{attribute 'GeneratedUsingTerminal: EK1100-0000-0018'}
{attribute addProperty BoxType "EK1100-0000-0018"}
{attribute addProperty Id "Beckhoff_EL73xxEK1122Beckhoff_EL73xxEK1122_D359B3E92A_0001_EL7332_0000_0016EL7332_B885ACFD38A_0002_EL7332_0000_0017EL7332_B885ACFD38A_0003_EL7332_0000_0018EL7332_B885ACFD38A_0004_EL7332_0000_0019EL7332_B885ACFD38A_0005_EL7332_0000_0020EL7332_B885ACFD38A_0006_EL7332_0000_0021EL7332_B885ACFD38A_0007_EL7332_0000_0022EL7332_B885ACFD38A_0008_EL7332_0000_0023EL7332_B885ACFD38A_0009_EL7332_0000_0024EL7332_B885ACFD38A_0010_EL7342_0000_0016EL7342_A970B60778A_0011_EL7342_0000_0017EL7342_A970B60778A_0012_EL7342_0000_0018EL7342_A970B60778A_0013_EL7342_0000_0019EL7342_A970B60778A_0014_EL7342_0000_0020EL7342_A970B60778A_0015_EL7342_0000_0021EL7342_A970B60778A_0016_EL7342_0000_0022EL7342_A970B60778A_0017_EL7342_0000_0023EL7342_C56E195380A_0018_EL7342_0035_0019EL7342_A970B60778A_0019_EL7342_0035_0020EL7342_A970B60778"}
{attribute addProperty CRC "3215524844"}
{attribute addProperty Size "1126"}
TYPE Beckhoff_EL73xx_BFA903EC EXTENDS EK1100_1FC0878B :
STRUCT
	{attribute addProperty Name "Beckhoff_EL73xxEK1122"}
	{attribute addProperty PreviousPort "Beckhoff EL73xx : B"}
	Beckhoff_EL73xxEK1122 : Beckhoff_EL73xxEK1122_D359B3E9;
	{attribute addProperty Name "A_0001_EL7332_0000_0016"}
	{attribute addProperty PreviousPort "Beckhoff EL73xxEK1122 : C"}
	A_0001_EL7332_0000_0016 : EL7332_B885ACFD;
	{attribute addProperty Name "A_0002_EL7332_0000_0017"}
	{attribute addProperty PreviousPort "A_0001(EL7332-0000-0016) : B"}
	A_0002_EL7332_0000_0017 : EL7332_B885ACFD;
	{attribute addProperty Name "A_0003_EL7332_0000_0018"}
	{attribute addProperty PreviousPort "A_0002(EL7332-0000-0017) : B"}
	A_0003_EL7332_0000_0018 : EL7332_B885ACFD;
	{attribute addProperty Name "A_0004_EL7332_0000_0019"}
	{attribute addProperty PreviousPort "A_0003(EL7332-0000-0018) : B"}
	A_0004_EL7332_0000_0019 : EL7332_B885ACFD;
	{attribute addProperty Name "A_0005_EL7332_0000_0020"}
	{attribute addProperty PreviousPort "A_0004(EL7332-0000-0019) : B"}
	A_0005_EL7332_0000_0020 : EL7332_B885ACFD;
	{attribute addProperty Name "A_0006_EL7332_0000_0021"}
	{attribute addProperty PreviousPort "A_0005(EL7332-0000-0020) : B"}
	A_0006_EL7332_0000_0021 : EL7332_B885ACFD;
	{attribute addProperty Name "A_0007_EL7332_0000_0022"}
	{attribute addProperty PreviousPort "A_0006(EL7332-0000-0021) : B"}
	A_0007_EL7332_0000_0022 : EL7332_B885ACFD;
	{attribute addProperty Name "A_0008_EL7332_0000_0023"}
	{attribute addProperty PreviousPort "A_0007(EL7332-0000-0022) : B"}
	A_0008_EL7332_0000_0023 : EL7332_B885ACFD;
	{attribute addProperty Name "A_0009_EL7332_0000_0024"}
	{attribute addProperty PreviousPort "A_0008(EL7332-0000-0023) : B"}
	A_0009_EL7332_0000_0024 : EL7332_B885ACFD;
	{attribute addProperty Name "A_0010_EL7342_0000_0016"}
	{attribute addProperty PreviousPort "A_0009(EL7332-0000-0024) : B"}
	A_0010_EL7342_0000_0016 : EL7342_A970B607;
	{attribute addProperty Name "A_0011_EL7342_0000_0017"}
	{attribute addProperty PreviousPort "A_0010(EL7342-0000-0016) : B"}
	A_0011_EL7342_0000_0017 : EL7342_A970B607;
	{attribute addProperty Name "A_0012_EL7342_0000_0018"}
	{attribute addProperty PreviousPort "A_0011(EL7342-0000-0017) : B"}
	A_0012_EL7342_0000_0018 : EL7342_A970B607;
	{attribute addProperty Name "A_0013_EL7342_0000_0019"}
	{attribute addProperty PreviousPort "A_0012(EL7342-0000-0018) : B"}
	A_0013_EL7342_0000_0019 : EL7342_A970B607;
	{attribute addProperty Name "A_0014_EL7342_0000_0020"}
	{attribute addProperty PreviousPort "A_0013(EL7342-0000-0019) : B"}
	A_0014_EL7342_0000_0020 : EL7342_A970B607;
	{attribute addProperty Name "A_0015_EL7342_0000_0021"}
	{attribute addProperty PreviousPort "A_0014(EL7342-0000-0020) : B"}
	A_0015_EL7342_0000_0021 : EL7342_A970B607;
	{attribute addProperty Name "A_0016_EL7342_0000_0022"}
	{attribute addProperty PreviousPort "A_0015(EL7342-0000-0021) : B"}
	A_0016_EL7342_0000_0022 : EL7342_A970B607;
	{attribute addProperty Name "A_0017_EL7342_0000_0023"}
	{attribute addProperty PreviousPort "A_0016(EL7342-0000-0022) : B"}
	A_0017_EL7342_0000_0023 : EL7342_C56E1953;
	{attribute addProperty Name "A_0018_EL7342_0035_0019"}
	{attribute addProperty PreviousPort "A_0017(EL7342-0000-0023) : B"}
	A_0018_EL7342_0035_0019 : EL7342_A970B607;
	{attribute addProperty Name "A_0019_EL7342_0035_0020"}
	{attribute addProperty PreviousPort "A_0018(EL7342-0035-0019) : B"}
	A_0019_EL7342_0035_0020 : EL7342_A970B607;
END_STRUCT
END_TYPE

(* stored: Version 1.2.0.0, ProductVersion 3.1.4024.9
   DUT Beckhoff_EL73xx_BFA903EC: Id {72c4eb52-9a7b-43d2-b25e-11665b4d98c7} *)
